(* Logix 5000 project; controller STAT 1756-L72 rev 20.12; software revision 20.04; part 6 of 34 *)
(* tags used below, declared in another part *)
   B11 : DINT[5];
   B15 : DINT[11];
   B3 : DINT[5];
   C5 : COUNTER[8];
   N17 : DINT[80];
   N7 : DINT[40];
   T10 : TIMER[30];
   T16 : TIMER[3];
   T4 : TIMER[30];
   def_fow_ecotec : BOOL;
   op010 : DINT;
   real : REAL;
   S_air_comp_Ecotech : REAL;
   S_cond_Ecotech : REAL;
   s_lvl_apu_feed_TK : DINT;
   s_lvl_filter_feed_TK : REAL;
   s_lvl_water_feed_TK : REAL;
   Scp_air_comp_Ecotech : SCP;
   Scp_cond_Ecotech : SCP;
   scp_lvl_apu_feed_TK : SCP;
   scp_lvl_filter_feed_TK : SCP;
   scp_lvl_water_feed_TK : SCP;
   toff_def_flow : TIMER;
   ton_run_eco : TIMER;
(* ECOTECH, continued *)

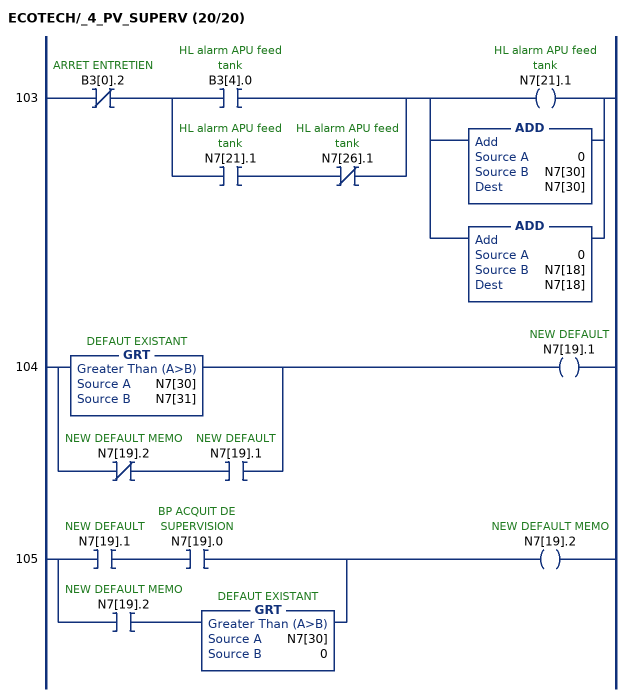
   [picture p46: ECOTECH/_4_PV_SUPERV rungs 103-105]
   103: XIO(B3[0].2)[XIC(B3[4].0) ,XIC(N7[21].1) XIO(N7[26].1) ][OTE(N7[21].1) ,ADD(0,N7[30],N7[30]) ,ADD(0,N7[18],N7[18]) ];
   104: [GRT(N7[30],N7[31]) ,XIO(N7[19].2) XIC(N7[19].1) ]OTE(N7[19].1);
   105: [XIC(N7[19].1) XIC(N7[19].0) ,XIC(N7[19].2) GRT(N7[30],0) ]OTE(N7[19].2);
END_ROUTINE

ROUTINE ECO_L4   (* ladder *)
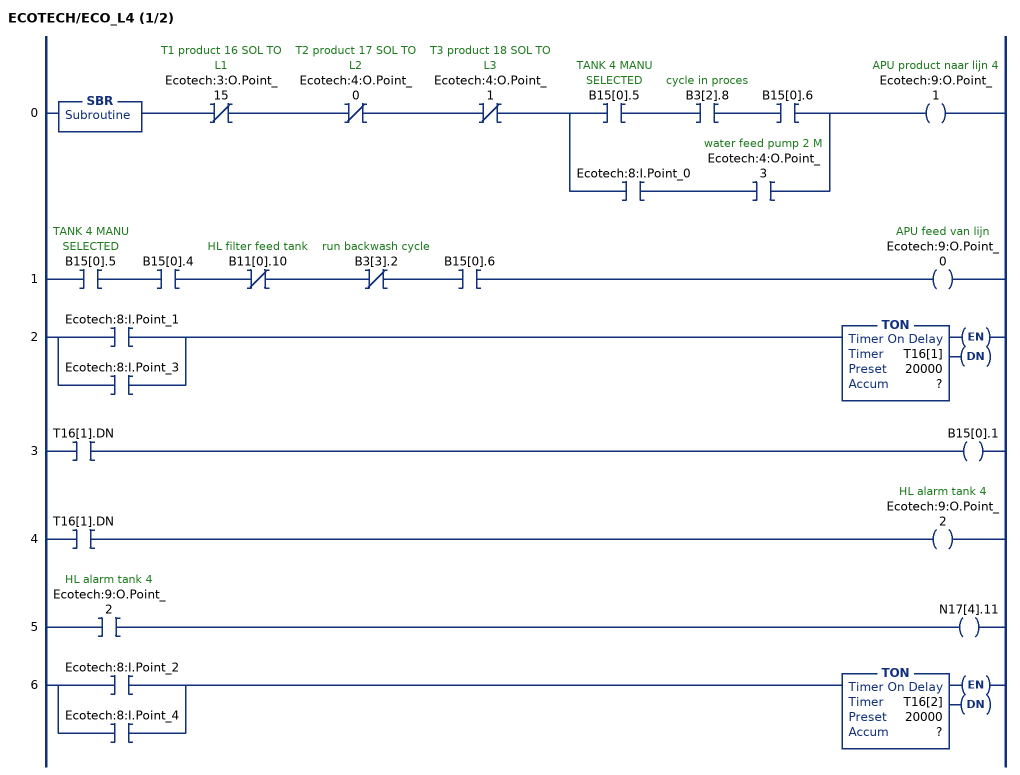
   0: SBR()XIO(Ecotech:3:O.Point_15)XIO(Ecotech:4:O.Point_0)XIO(Ecotech:4:O.Point_1)[XIC(B15[0].5) XIC(B3[2].8) XIC(B15[0].6) ,XIC(Ecotech:8:I.Point_0) XIC(Ecotech:4:O.Point_3) ]OTE(Ecotech:9:O.Point_1);
   1: XIC(B15[0].5)XIC(B15[0].4)XIO(B11[0].10)XIO(B3[3].2)XIC(B15[0].6)OTE(Ecotech:9:O.Point_0);
   2: [XIC(Ecotech:8:I.Point_1) ,XIC(Ecotech:8:I.Point_3) ]TON(T16[1],?,?);
   3: XIC(T16[1].DN)OTE(B15[0].1);
   4: XIC(T16[1].DN)OTE(Ecotech:9:O.Point_2);
   5: XIC(Ecotech:9:O.Point_2)OTE(N17[4].11);
   6: [XIC(Ecotech:8:I.Point_2) ,XIC(Ecotech:8:I.Point_4) ]TON(T16[2],?,?);
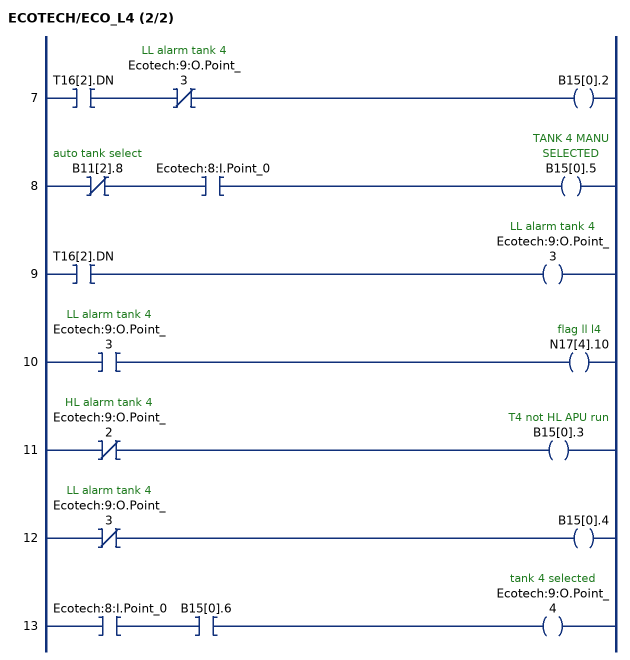
   7: XIC(T16[2].DN)XIO(Ecotech:9:O.Point_3)OTE(B15[0].2);
   8: XIO(B11[2].8)XIC(Ecotech:8:I.Point_0)OTE(B15[0].5);
   9: XIC(T16[2].DN)OTE(Ecotech:9:O.Point_3);
   10: XIC(Ecotech:9:O.Point_3)OTE(N17[4].10);
   11: XIO(Ecotech:9:O.Point_2)OTE(B15[0].3);
   12: XIO(Ecotech:9:O.Point_3)OTE(B15[0].4);
   13: XIC(Ecotech:8:I.Point_0)XIC(B15[0].6)OTE(Ecotech:9:O.Point_4);
END_ROUTINE

ROUTINE ECO_Main   (* ladder *)
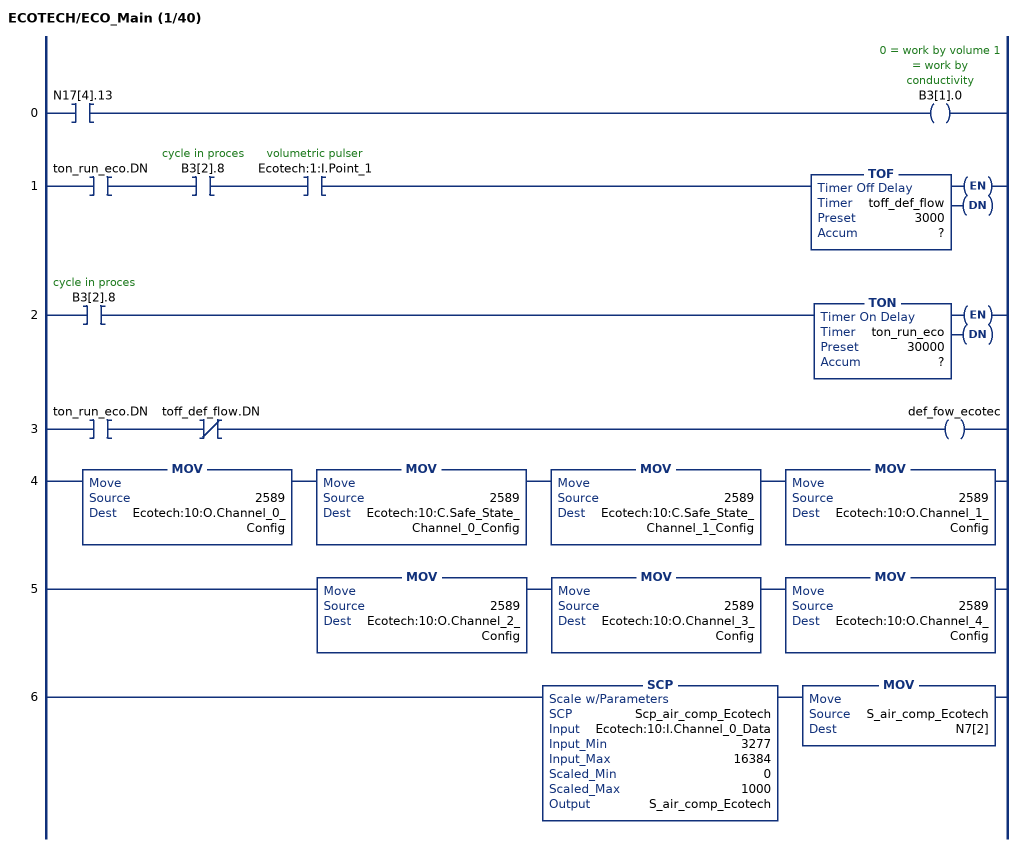
   0: XIC(N17[4].13)OTE(B3[1].0);
   1: XIC(ton_run_eco.DN)XIC(B3[2].8)XIC(Ecotech:1:I.Point_1)TOF(toff_def_flow,?,?);
   2: XIC(B3[2].8)TON(ton_run_eco,?,?);
   3: XIC(ton_run_eco.DN)XIO(toff_def_flow.DN)OTE(def_fow_ecotec);
   4: MOV(2589,Ecotech:10:O.Channel_0_Config)MOV(2589,Ecotech:10:C.Safe_State_Channel_0_Config)MOV(2589,Ecotech:10:C.Safe_State_Channel_1_Config)MOV(2589,Ecotech:10:O.Channel_1_Config);
   5: MOV(2589,Ecotech:10:O.Channel_2_Config)MOV(2589,Ecotech:10:O.Channel_3_Config)MOV(2589,Ecotech:10:O.Channel_4_Config);
   6: SCP(Scp_air_comp_Ecotech,Ecotech:10:I.Channel_0_Data,3277,16384,0,1000,S_air_comp_Ecotech)MOV(S_air_comp_Ecotech,N7[2]);
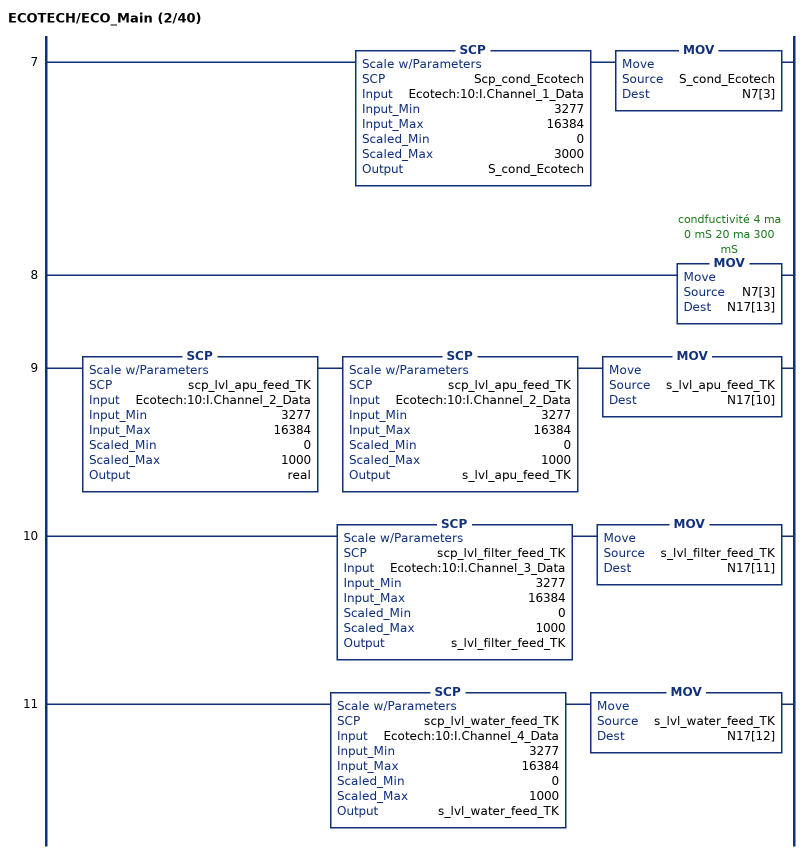
   7: SCP(Scp_cond_Ecotech,Ecotech:10:I.Channel_1_Data,3277,16384,0,3000,S_cond_Ecotech)MOV(S_cond_Ecotech,N7[3]);
   8: MOV(N7[3],N17[13]);
   9: SCP(scp_lvl_apu_feed_TK,Ecotech:10:I.Channel_2_Data,3277,16384,0,1000,real)SCP(scp_lvl_apu_feed_TK,Ecotech:10:I.Channel_2_Data,3277,16384,0,1000,s_lvl_apu_feed_TK)MOV(s_lvl_apu_feed_TK,N17[10]);
   10: SCP(scp_lvl_filter_feed_TK,Ecotech:10:I.Channel_3_Data,3277,16384,0,1000,s_lvl_filter_feed_TK)MOV(s_lvl_filter_feed_TK,N17[11]);
   11: SCP(scp_lvl_water_feed_TK,Ecotech:10:I.Channel_4_Data,3277,16384,0,1000,s_lvl_water_feed_TK)MOV(s_lvl_water_feed_TK,N17[12]);
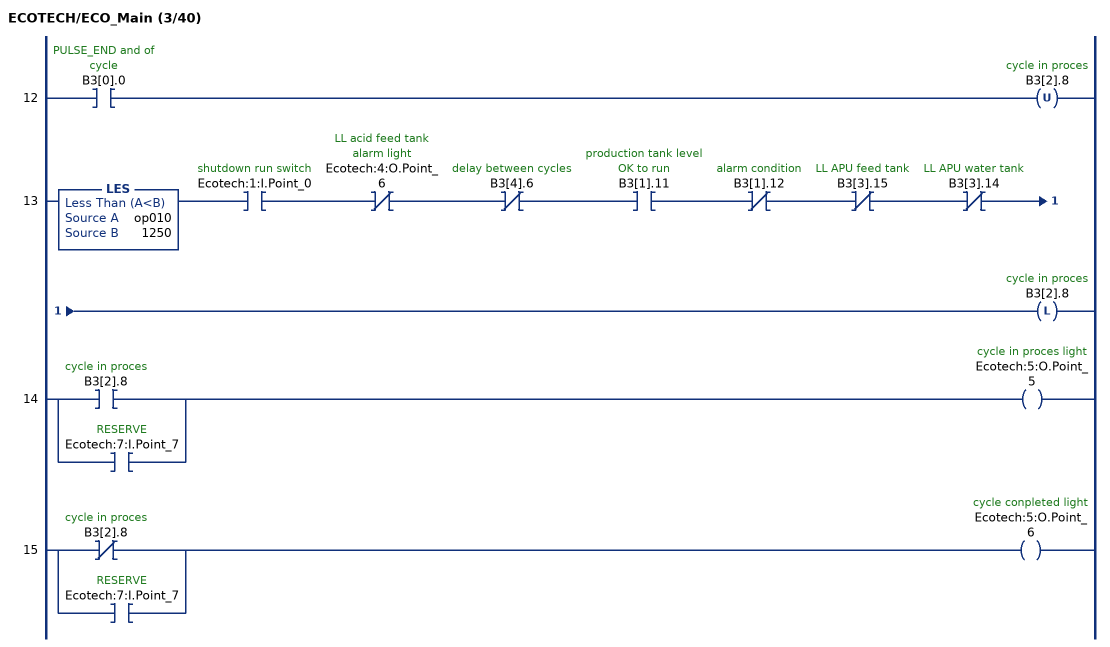
   12: XIC(B3[0].0)OTU(B3[2].8);
   13: LES(op010,1250)XIC(Ecotech:1:I.Point_0)XIO(Ecotech:4:O.Point_6)XIO(B3[4].6)XIC(B3[1].11)XIO(B3[1].12)XIO(B3[3].15)XIO(B3[3].14)OTL(B3[2].8);
   14: [XIC(B3[2].8) ,XIC(Ecotech:7:I.Point_7) ]OTE(Ecotech:5:O.Point_5);
   15: [XIO(B3[2].8) ,XIC(Ecotech:7:I.Point_7) ]OTE(Ecotech:5:O.Point_6);
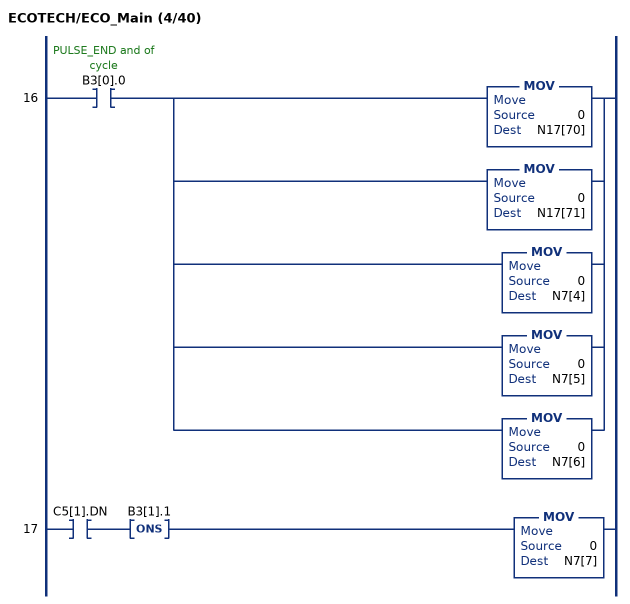
   16: XIC(B3[0].0)[MOV(0,N17[70]) ,MOV(0,N17[71]) ,MOV(0,N7[4]) ,MOV(0,N7[5]) ,MOV(0,N7[6]) ];
   17: XIC(C5[1].DN)ONS(B3[1].1)MOV(0,N7[7]);
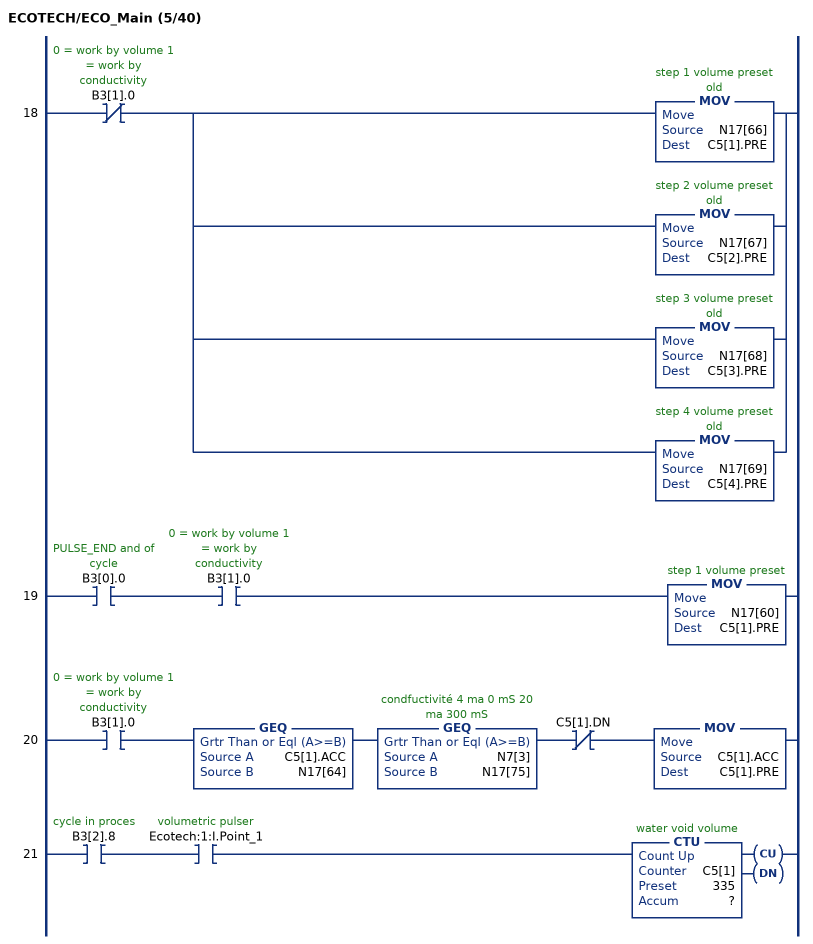
   18: XIO(B3[1].0)[MOV(N17[66],C5[1].PRE) ,MOV(N17[67],C5[2].PRE) ,MOV(N17[68],C5[3].PRE) ,MOV(N17[69],C5[4].PRE) ];
   19: XIC(B3[0].0)XIC(B3[1].0)MOV(N17[60],C5[1].PRE);
   20: XIC(B3[1].0)GEQ(C5[1].ACC,N17[64])GEQ(N7[3],N17[75])XIO(C5[1].DN)MOV(C5[1].ACC,C5[1].PRE);
   21: XIC(B3[2].8)XIC(Ecotech:1:I.Point_1)CTU(C5[1],?,?);
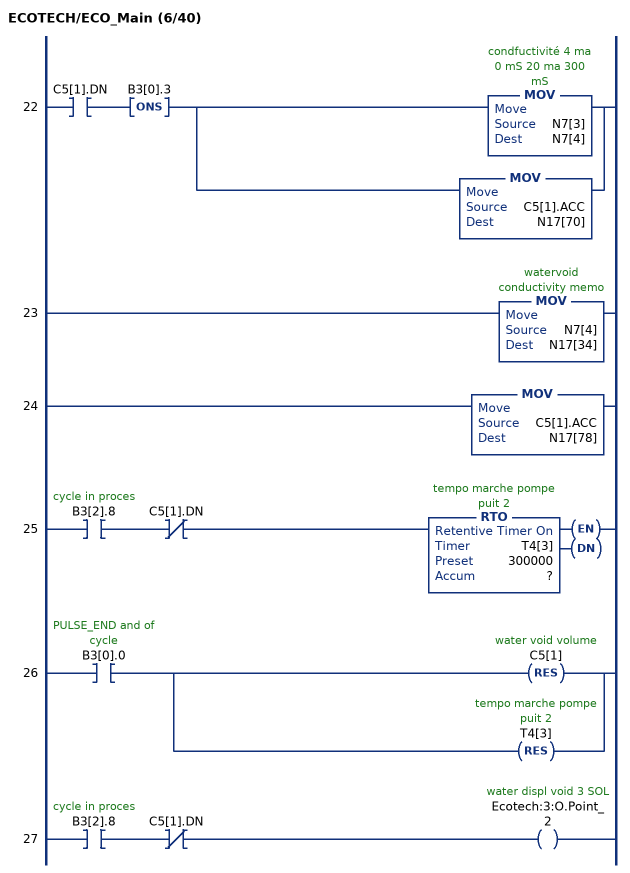
   22: XIC(C5[1].DN)ONS(B3[0].3)[MOV(N7[3],N7[4]) ,MOV(C5[1].ACC,N17[70]) ];
   23: MOV(N7[4],N17[34]);
   24: MOV(C5[1].ACC,N17[78]);
   25: XIC(B3[2].8)XIO(C5[1].DN)RTO(T4[3],?,?);
   26: XIC(B3[0].0)[RES(C5[1]) ,RES(T4[3]) ];
   27: XIC(B3[2].8)XIO(C5[1].DN)OTE(Ecotech:3:O.Point_2);
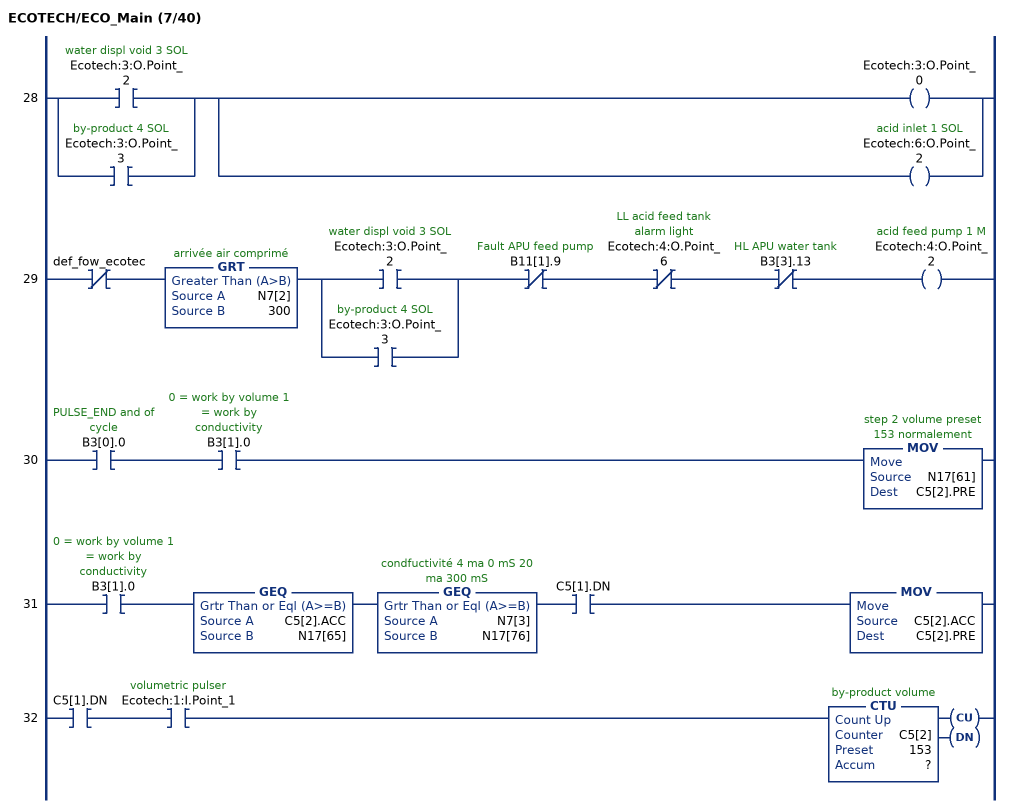
   28: [XIC(Ecotech:3:O.Point_2) ,XIC(Ecotech:3:O.Point_3) ][OTE(Ecotech:3:O.Point_0) ,OTE(Ecotech:6:O.Point_2) ];
   29: XIO(def_fow_ecotec)GRT(N7[2],300)[XIC(Ecotech:3:O.Point_2) ,XIC(Ecotech:3:O.Point_3) ]XIO(B11[1].9)XIO(Ecotech:4:O.Point_6)XIO(B3[3].13)OTE(Ecotech:4:O.Point_2);
   30: XIC(B3[0].0)XIC(B3[1].0)MOV(N17[61],C5[2].PRE);
   31: XIC(B3[1].0)GEQ(C5[2].ACC,N17[65])GEQ(N7[3],N17[76])XIC(C5[1].DN)MOV(C5[2].ACC,C5[2].PRE);
   32: XIC(C5[1].DN)XIC(Ecotech:1:I.Point_1)CTU(C5[2],?,?);
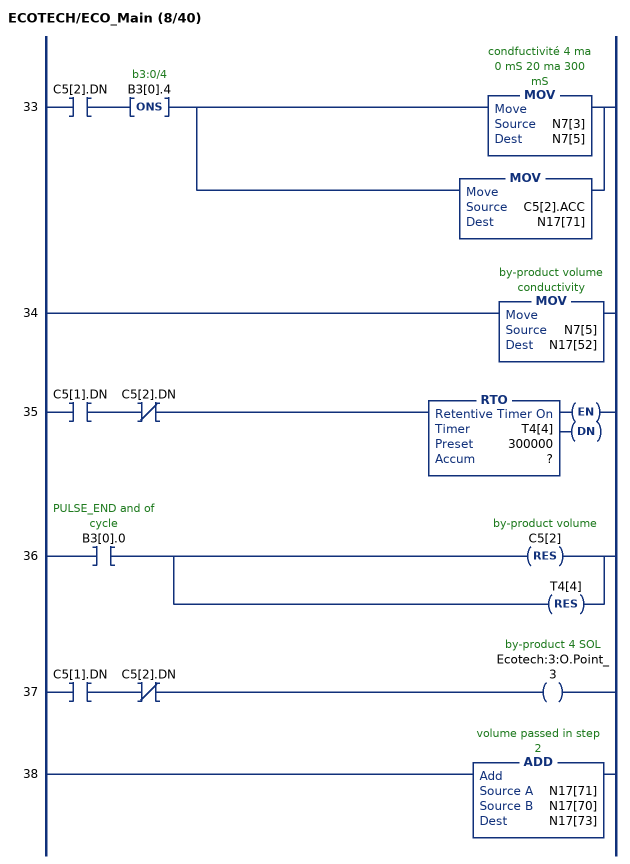
   33: XIC(C5[2].DN)ONS(B3[0].4)[MOV(N7[3],N7[5]) ,MOV(C5[2].ACC,N17[71]) ];
   34: MOV(N7[5],N17[52]);
   35: XIC(C5[1].DN)XIO(C5[2].DN)RTO(T4[4],?,?);
   36: XIC(B3[0].0)[RES(C5[2]) ,RES(T4[4]) ];
   37: XIC(C5[1].DN)XIO(C5[2].DN)OTE(Ecotech:3:O.Point_3);
   38: ADD(N17[71],N17[70],N17[73]);
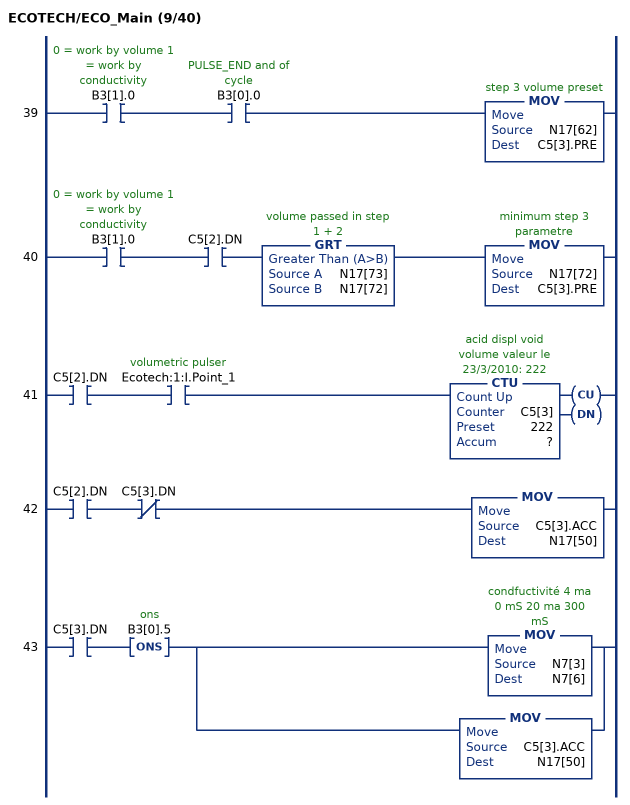
   39: XIC(B3[1].0)XIC(B3[0].0)MOV(N17[62],C5[3].PRE);
   40: XIC(B3[1].0)XIC(C5[2].DN)GRT(N17[73],N17[72])MOV(N17[72],C5[3].PRE);
   41: XIC(C5[2].DN)XIC(Ecotech:1:I.Point_1)CTU(C5[3],?,?);
   42: XIC(C5[2].DN)XIO(C5[3].DN)MOV(C5[3].ACC,N17[50]);
   43: XIC(C5[3].DN)ONS(B3[0].5)[MOV(N7[3],N7[6]) ,MOV(C5[3].ACC,N17[50]) ];
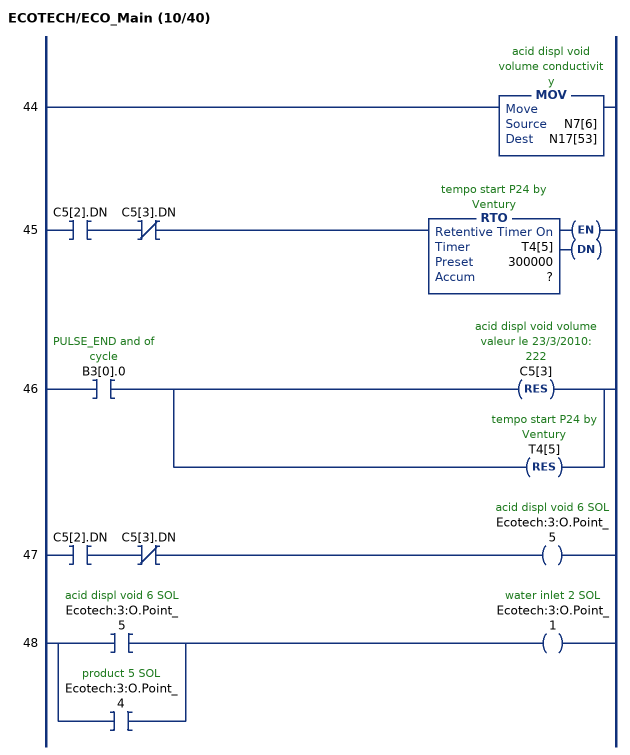
   44: MOV(N7[6],N17[53]);
   45: XIC(C5[2].DN)XIO(C5[3].DN)RTO(T4[5],?,?);
   46: XIC(B3[0].0)[RES(C5[3]) ,RES(T4[5]) ];
   47: XIC(C5[2].DN)XIO(C5[3].DN)OTE(Ecotech:3:O.Point_5);
   48: [XIC(Ecotech:3:O.Point_5) ,XIC(Ecotech:3:O.Point_4) ]OTE(Ecotech:3:O.Point_1);
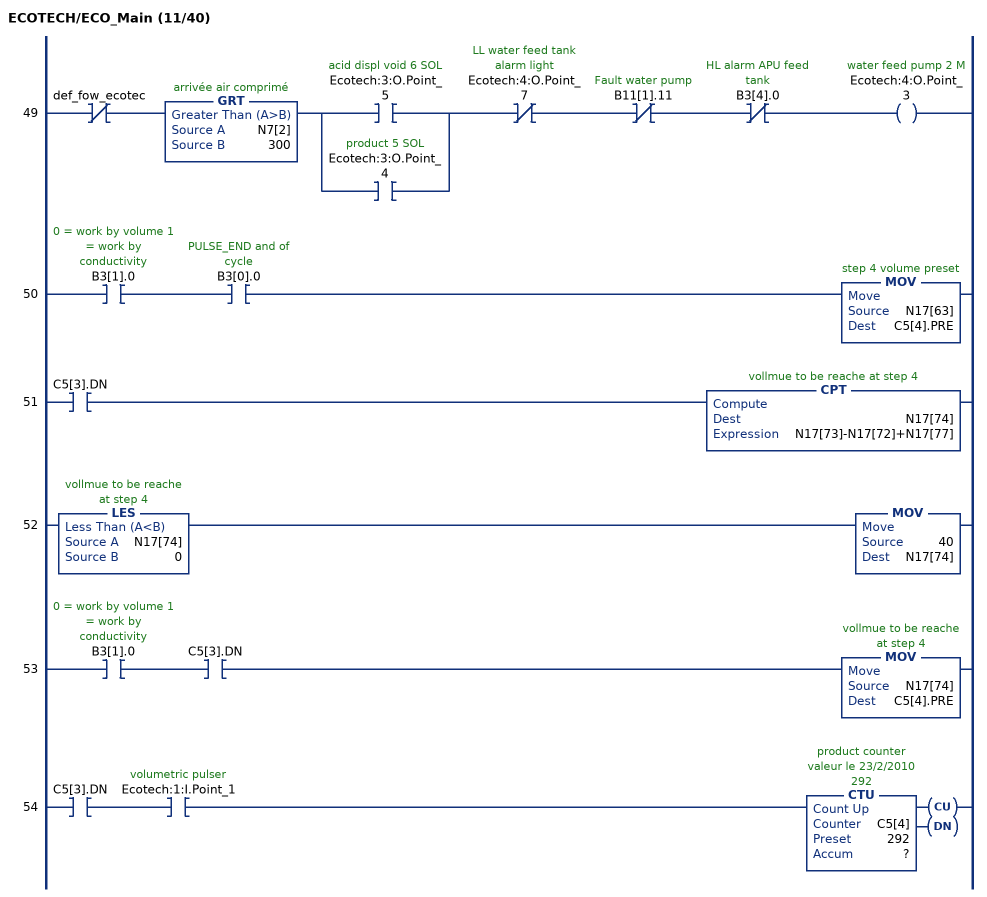
   49: XIO(def_fow_ecotec)GRT(N7[2],300)[XIC(Ecotech:3:O.Point_5) ,XIC(Ecotech:3:O.Point_4) ]XIO(Ecotech:4:O.Point_7)XIO(B11[1].11)XIO(B3[4].0)OTE(Ecotech:4:O.Point_3);
   50: XIC(B3[1].0)XIC(B3[0].0)MOV(N17[63],C5[4].PRE);
   51: XIC(C5[3].DN)CPT(N17[74],N17[73]-N17[72]+N17[77]);
   52: LES(N17[74],0)MOV(40,N17[74]);
   53: XIC(B3[1].0)XIC(C5[3].DN)MOV(N17[74],C5[4].PRE);
   54: XIC(C5[3].DN)XIC(Ecotech:1:I.Point_1)CTU(C5[4],?,?);
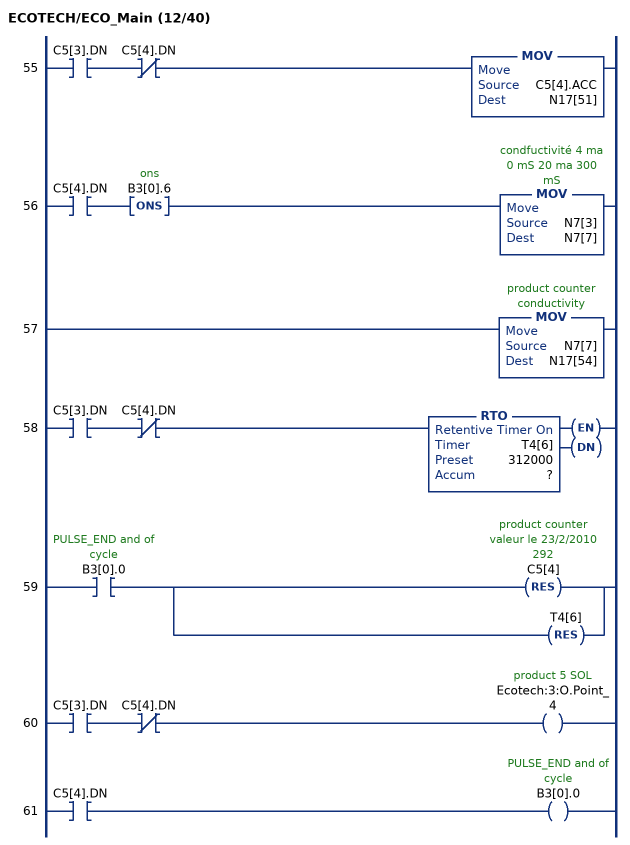
   55: XIC(C5[3].DN)XIO(C5[4].DN)MOV(C5[4].ACC,N17[51]);
   56: XIC(C5[4].DN)ONS(B3[0].6)MOV(N7[3],N7[7]);
   57: MOV(N7[7],N17[54]);
   58: XIC(C5[3].DN)XIO(C5[4].DN)RTO(T4[6],?,?);
   59: XIC(B3[0].0)[RES(C5[4]) ,RES(T4[6]) ];
   60: XIC(C5[3].DN)XIO(C5[4].DN)OTE(Ecotech:3:O.Point_4);
   61: XIC(C5[4].DN)OTE(B3[0].0);
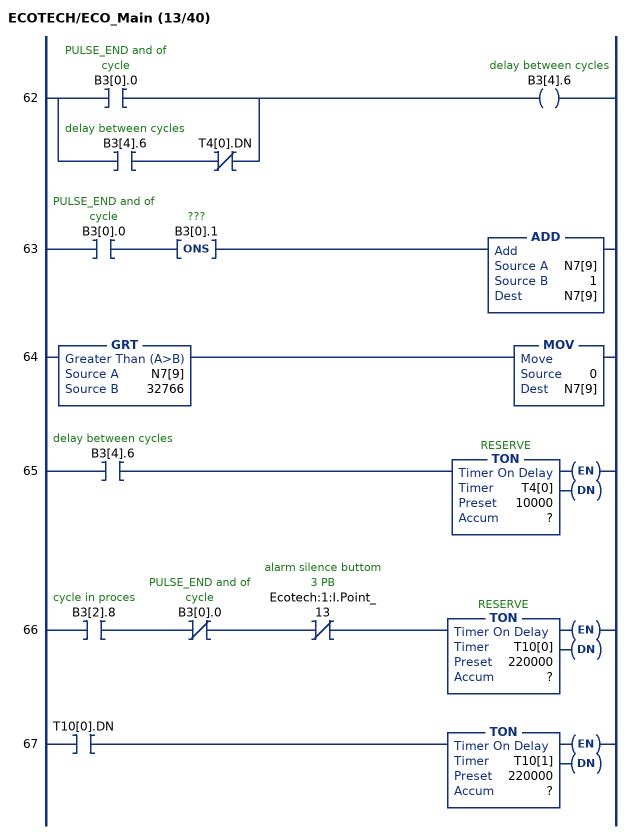
   62: [XIC(B3[0].0) ,XIC(B3[4].6) XIO(T4[0].DN) ]OTE(B3[4].6);
   63: XIC(B3[0].0)ONS(B3[0].1)ADD(N7[9],1,N7[9]);
   64: GRT(N7[9],32766)MOV(0,N7[9]);
   65: XIC(B3[4].6)TON(T4[0],?,?);
   66: XIC(B3[2].8)XIO(B3[0].0)XIO(Ecotech:1:I.Point_13)TON(T10[0],?,?);
   67: XIC(T10[0].DN)TON(T10[1],?,?);
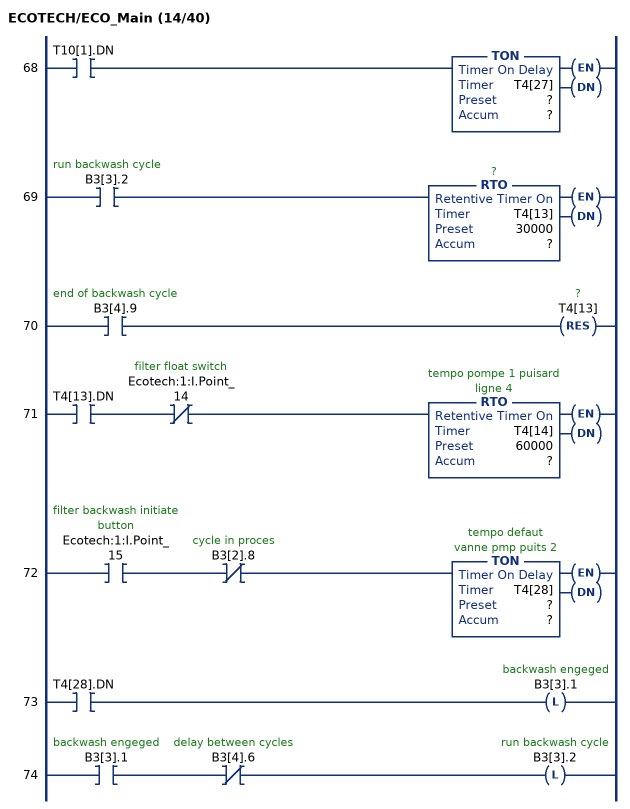
   68: XIC(T10[1].DN)TON(T4[27],?,?);
   69: XIC(B3[3].2)RTO(T4[13],?,?);
   70: XIC(B3[4].9)RES(T4[13]);
   71: XIC(T4[13].DN)XIO(Ecotech:1:I.Point_14)RTO(T4[14],?,?);
   72: XIC(Ecotech:1:I.Point_15)XIO(B3[2].8)TON(T4[28],?,?);
   73: XIC(T4[28].DN)OTL(B3[3].1);
   74: XIC(B3[3].1)XIO(B3[4].6)OTL(B3[3].2);
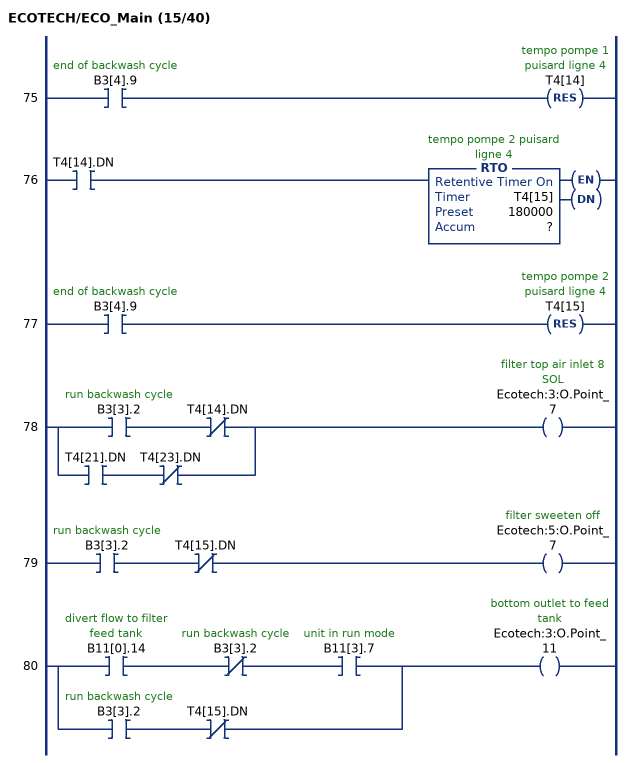
   75: XIC(B3[4].9)RES(T4[14]);
   76: XIC(T4[14].DN)RTO(T4[15],?,?);
   77: XIC(B3[4].9)RES(T4[15]);
   78: [XIC(B3[3].2) XIO(T4[14].DN) ,XIC(T4[21].DN) XIO(T4[23].DN) ]OTE(Ecotech:3:O.Point_7);
   79: XIC(B3[3].2)XIO(T4[15].DN)OTE(Ecotech:5:O.Point_7);
   80: [XIC(B11[0].14) XIO(B3[3].2) XIC(B11[3].7) ,XIC(B3[3].2) XIO(T4[15].DN) ]OTE(Ecotech:3:O.Point_11);
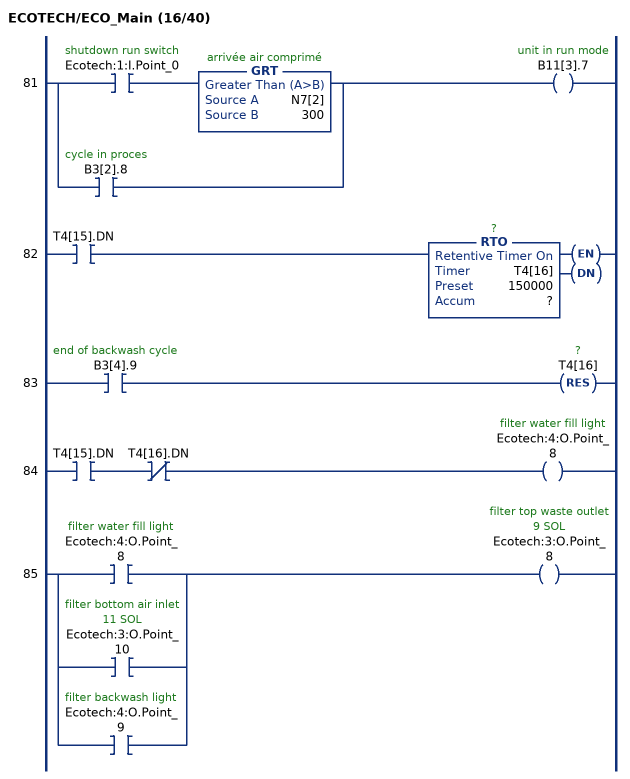
   81: [XIC(Ecotech:1:I.Point_0) GRT(N7[2],300) ,XIC(B3[2].8) ]OTE(B11[3].7);
   82: XIC(T4[15].DN)RTO(T4[16],?,?);
   83: XIC(B3[4].9)RES(T4[16]);
   84: XIC(T4[15].DN)XIO(T4[16].DN)OTE(Ecotech:4:O.Point_8);
   85: [XIC(Ecotech:4:O.Point_8) ,XIC(Ecotech:3:O.Point_10) ,XIC(Ecotech:4:O.Point_9) ]OTE(Ecotech:3:O.Point_8);
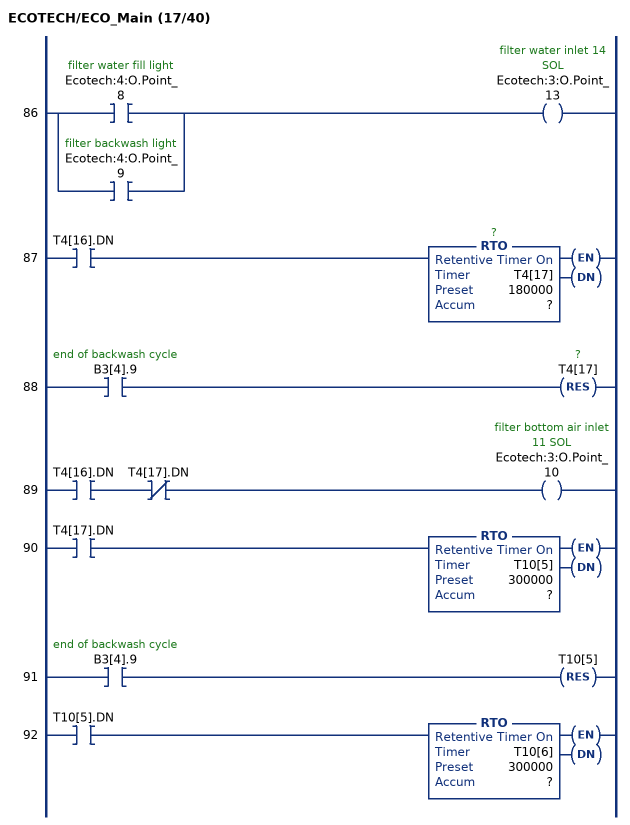
   86: [XIC(Ecotech:4:O.Point_8) ,XIC(Ecotech:4:O.Point_9) ]OTE(Ecotech:3:O.Point_13);
   87: XIC(T4[16].DN)RTO(T4[17],?,?);
   88: XIC(B3[4].9)RES(T4[17]);
   89: XIC(T4[16].DN)XIO(T4[17].DN)OTE(Ecotech:3:O.Point_10);
   90: XIC(T4[17].DN)RTO(T10[5],?,?);
   91: XIC(B3[4].9)RES(T10[5]);
   92: XIC(T10[5].DN)RTO(T10[6],?,?);
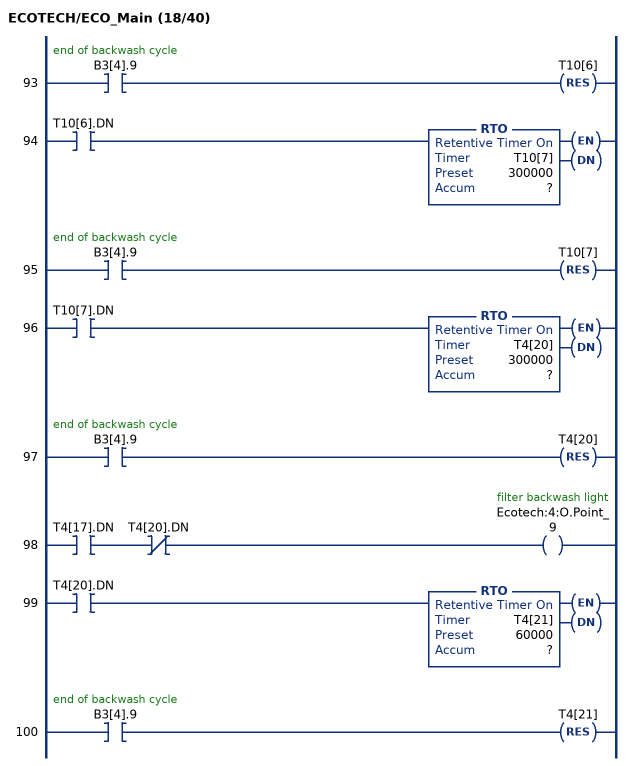
   93: XIC(B3[4].9)RES(T10[6]);
   94: XIC(T10[6].DN)RTO(T10[7],?,?);
   95: XIC(B3[4].9)RES(T10[7]);
   96: XIC(T10[7].DN)RTO(T4[20],?,?);
   97: XIC(B3[4].9)RES(T4[20]);
   98: XIC(T4[17].DN)XIO(T4[20].DN)OTE(Ecotech:4:O.Point_9);
   99: XIC(T4[20].DN)RTO(T4[21],?,?);
   100: XIC(B3[4].9)RES(T4[21]);
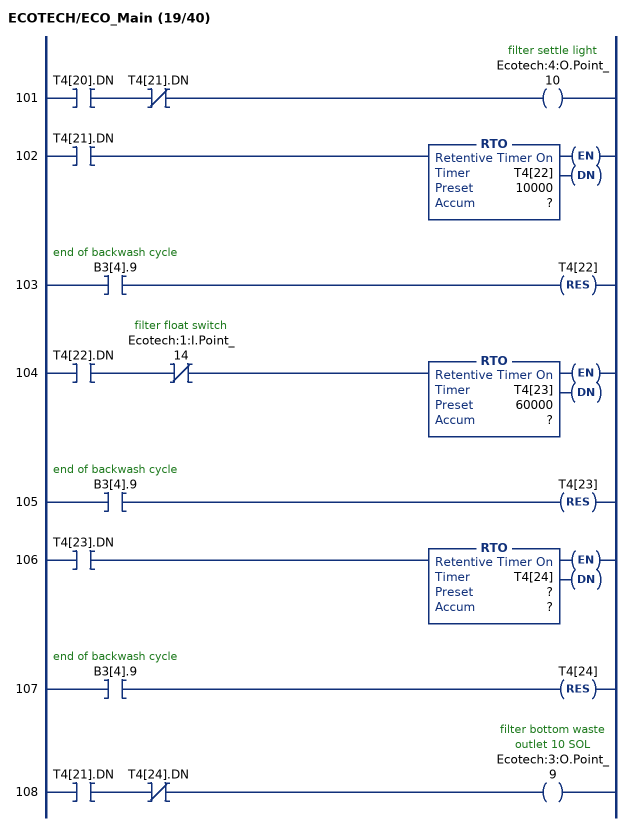
   101: XIC(T4[20].DN)XIO(T4[21].DN)OTE(Ecotech:4:O.Point_10);
   102: XIC(T4[21].DN)RTO(T4[22],?,?);
   103: XIC(B3[4].9)RES(T4[22]);
   104: XIC(T4[22].DN)XIO(Ecotech:1:I.Point_14)RTO(T4[23],?,?);
   105: XIC(B3[4].9)RES(T4[23]);
   106: XIC(T4[23].DN)RTO(T4[24],?,?);
   107: XIC(B3[4].9)RES(T4[24]);
   108: XIC(T4[21].DN)XIO(T4[24].DN)OTE(Ecotech:3:O.Point_9);
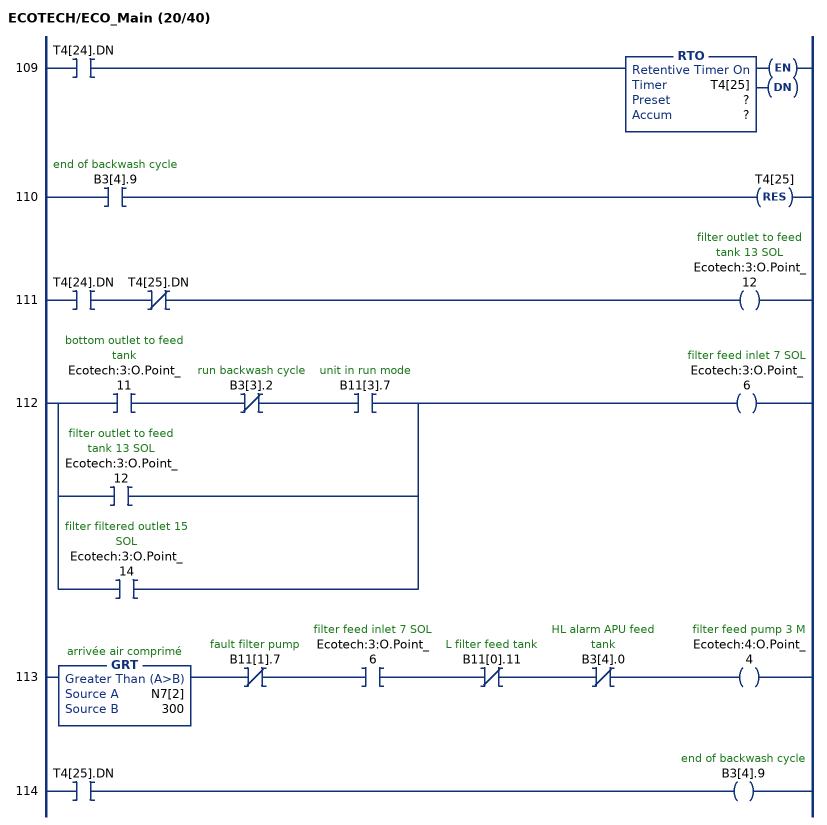
   109: XIC(T4[24].DN)RTO(T4[25],?,?);
   110: XIC(B3[4].9)RES(T4[25]);
   111: XIC(T4[24].DN)XIO(T4[25].DN)OTE(Ecotech:3:O.Point_12);
   112: [XIC(Ecotech:3:O.Point_11) XIO(B3[3].2) XIC(B11[3].7) ,XIC(Ecotech:3:O.Point_12) ,XIC(Ecotech:3:O.Point_14) ]OTE(Ecotech:3:O.Point_6);
   113: GRT(N7[2],300)XIO(B11[1].7)XIC(Ecotech:3:O.Point_6)XIO(B11[0].11)XIO(B3[4].0)OTE(Ecotech:4:O.Point_4);
   114: XIC(T4[25].DN)OTE(B3[4].9);
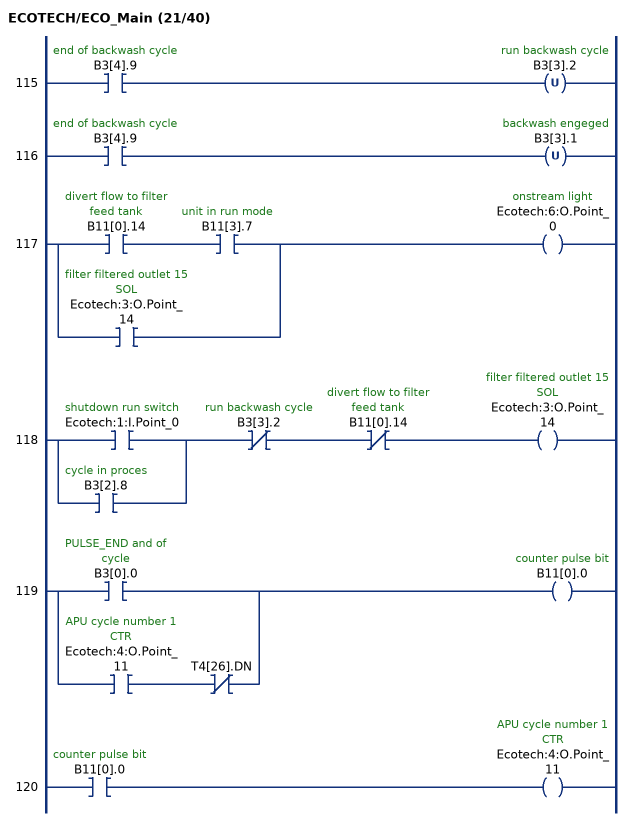
   115: XIC(B3[4].9)OTU(B3[3].2);
   116: XIC(B3[4].9)OTU(B3[3].1);
   117: [XIC(B11[0].14) XIC(B11[3].7) ,XIC(Ecotech:3:O.Point_14) ]OTE(Ecotech:6:O.Point_0);
   118: [XIC(Ecotech:1:I.Point_0) ,XIC(B3[2].8) ]XIO(B3[3].2)XIO(B11[0].14)OTE(Ecotech:3:O.Point_14);
   119: [XIC(B3[0].0) ,XIC(Ecotech:4:O.Point_11) XIO(T4[26].DN) ]OTE(B11[0].0);
   120: XIC(B11[0].0)OTE(Ecotech:4:O.Point_11);
